% RSLogix 500 project AGEOVEN_NEW19.RSS, saved by version 12.00.00.00 %
PROJECT "UNTITLED"    % processor: type code 47 %

PROGRAM FILES
  LAD 2   3 rungs
  LAD 3   11 rungs
  LAD 4   8 rungs

DATA FILES
  O0 OUTPUT  9 elements
  I1 INPUT  9 elements
  S2 STATUS  83 elements
  B3 BINARY  1 elements
  T4 TIMER  1 elements
  C5 COUNTER  1 elements
  R6 CONTROL  1 elements
  N7 INTEGER  25 elements
  F8 FLOAT  2 elements

LADDER 2
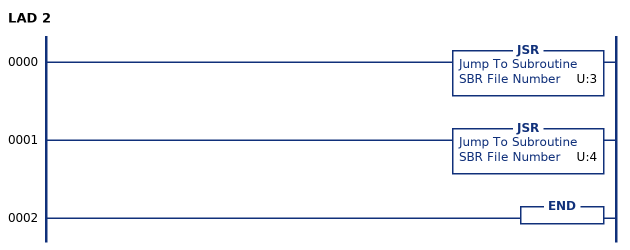
% Rung: 0 %
SOR JSR U:3 EOR
% Rung: 1 %
SOR JSR U:4 EOR
% Rung: 2 %
SOR END EOR

LADDER 3
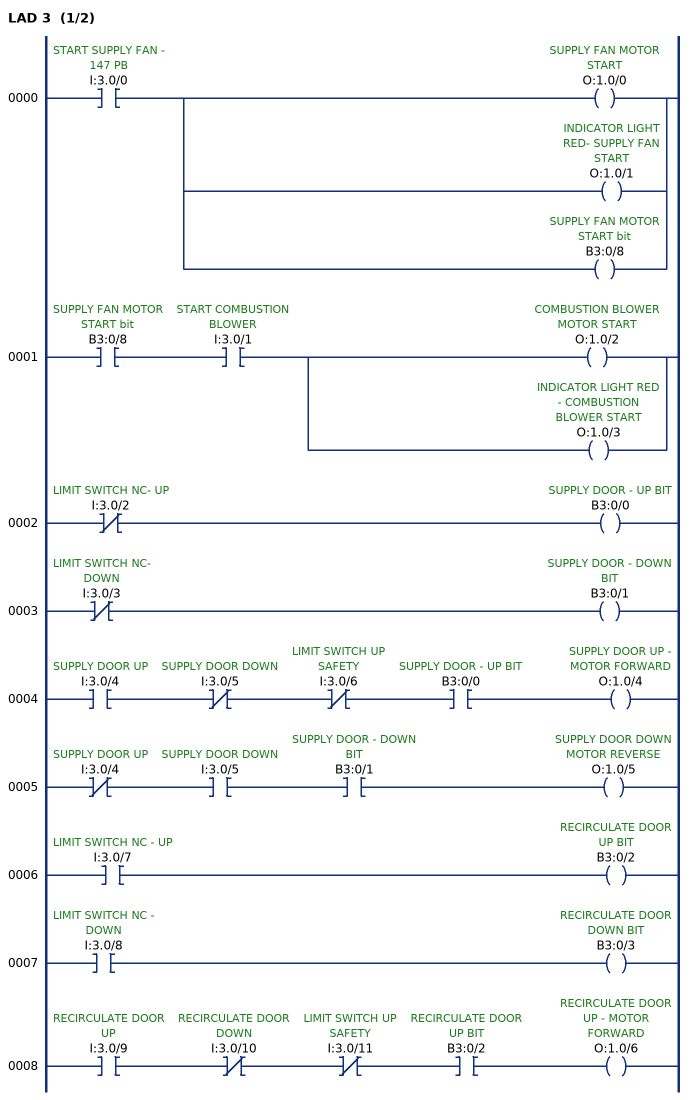
% Rung: 0 %
SOR XIC I:3.0/0 BST OTE O:1.0/0 NXB OTE O:1.0/1 NXB OTE B3:0/8 BND EOR
%   I:3.0/0  "START SUPPLY FAN - 147 PB" %
%   O:1.0/0  "SUPPLY FAN MOTOR START" %
%   O:1.0/1  "INDICATOR LIGHT RED- SUPPLY FAN START" %
%   B3:0/8  "SUPPLY FAN MOTOR START bit" %
% Rung: 1 %
SOR XIC B3:0/8 XIC I:3.0/1 BST OTE O:1.0/2 NXB OTE O:1.0/3 BND EOR
%   B3:0/8  "SUPPLY FAN MOTOR START bit" %
%   I:3.0/1  "START COMBUSTION BLOWER" %
%   O:1.0/2  "COMBUSTION BLOWER MOTOR START" %
%   O:1.0/3  "INDICATOR LIGHT RED - COMBUSTION BLOWER START" %
% Rung: 2 %  % edit flag set %
SOR XIO I:3.0/2 OTE B3:0/0 EOR
%   I:3.0/2  "LIMIT SWITCH NC- UP" %
%   B3:0/0  "SUPPLY DOOR - UP BIT" %
% Rung: 3 %  % edit flag set %
SOR XIO I:3.0/3 OTE B3:0/1 EOR
%   I:3.0/3  "LIMIT SWITCH NC- DOWN" %
%   B3:0/1  "SUPPLY DOOR - DOWN BIT" %
% Rung: 4 %
SOR XIC I:3.0/4 XIO I:3.0/5 XIO I:3.0/6 XIC B3:0/0 OTE O:1.0/4 EOR
%   I:3.0/4  "SUPPLY DOOR UP" %
%   I:3.0/5  "SUPPLY DOOR DOWN" %
%   I:3.0/6  "LIMIT SWITCH UP SAFETY" %
%   B3:0/0  "SUPPLY DOOR - UP BIT" %
%   O:1.0/4  "SUPPLY DOOR UP - MOTOR FORWARD" %
% Rung: 5 %
SOR XIO I:3.0/4 XIC I:3.0/5 XIC B3:0/1 OTE O:1.0/5 EOR
%   I:3.0/4  "SUPPLY DOOR UP" %
%   I:3.0/5  "SUPPLY DOOR DOWN" %
%   B3:0/1  "SUPPLY DOOR - DOWN BIT" %
%   O:1.0/5  "SUPPLY DOOR DOWN MOTOR REVERSE" %
% Rung: 6 %
SOR XIC I:3.0/7 OTE B3:0/2 EOR
%   I:3.0/7  "LIMIT SWITCH NC - UP" %
%   B3:0/2  "RECIRCULATE DOOR UP BIT" %
% Rung: 7 %
SOR XIC I:3.0/8 OTE B3:0/3 EOR
%   I:3.0/8  "LIMIT SWITCH NC - DOWN" %
%   B3:0/3  "RECIRCULATE DOOR DOWN BIT" %
% Rung: 8 %
SOR XIC I:3.0/9 XIO I:3.0/10 XIO I:3.0/11 XIC B3:0/2 OTE O:1.0/6 EOR
%   I:3.0/9  "RECIRCULATE DOOR UP" %
%   I:3.0/10  "RECIRCULATE DOOR DOWN" %
%   I:3.0/11  "LIMIT SWITCH UP SAFETY" %
%   B3:0/2  "RECIRCULATE DOOR UP BIT" %
%   O:1.0/6  "RECIRCULATE DOOR UP - MOTOR FORWARD" %

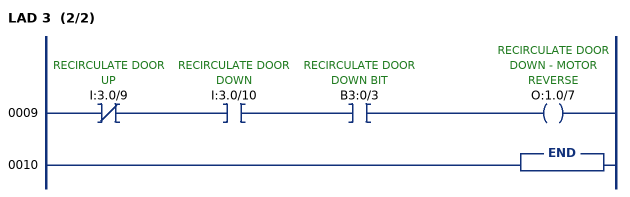
% Rung: 9 %
SOR XIO I:3.0/9 XIC I:3.0/10 XIC B3:0/3 OTE O:1.0/7 EOR
%   I:3.0/9  "RECIRCULATE DOOR UP" %
%   I:3.0/10  "RECIRCULATE DOOR DOWN" %
%   B3:0/3  "RECIRCULATE DOOR DOWN BIT" %
%   O:1.0/7  "RECIRCULATE DOOR DOWN - MOTOR REVERSE" %
% Rung: 10 %
SOR END EOR

LADDER 4
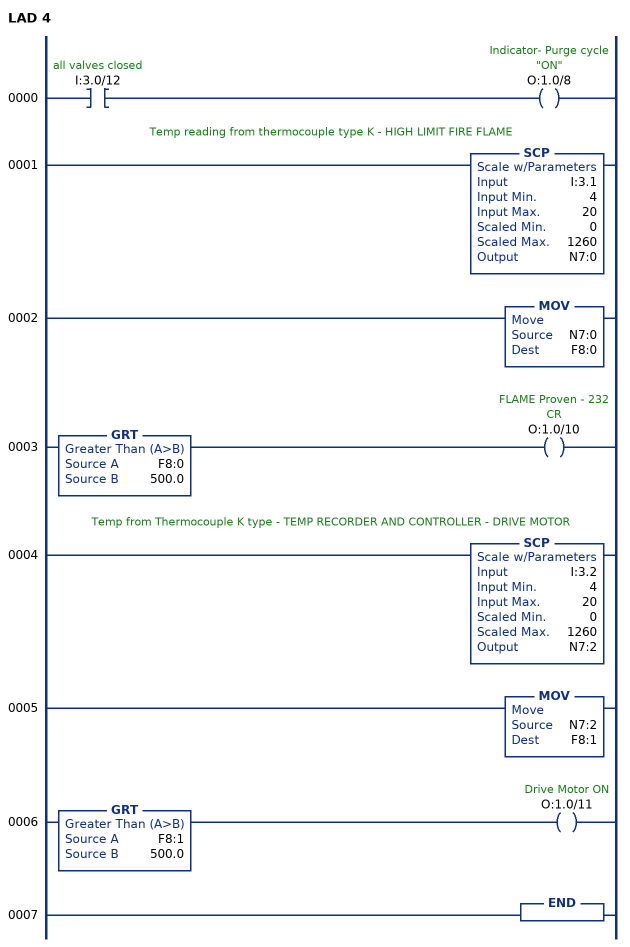
% Rung: 0 %
SOR XIC I:3.0/12 OTE O:1.0/8 EOR
%   I:3.0/12  "all valves closed" %
%   O:1.0/8  "Indicator- Purge cycle "ON"" %
% Rung: 1 %
% Temp reading from thermocouple type K - HIGH LIMIT FIRE FLAME %
SOR SCP I:3.1 4 20 0 1260 N7:0 EOR
%   I:3.1  "Thermocouple for tempretaure control" %
% Rung: 2 %
SOR MOV N7:0 F8:0 EOR
% Rung: 3 %
SOR GRT F8:0 500.0 OTE O:1.0/10 EOR
%   O:1.0/10  "FLAME Proven - 232 CR" %
% Rung: 4 %
% Temp from Thermocouple K type - TEMP RECORDER AND CONTROLLER - DRIVE MOTOR %
SOR SCP I:3.2 4 20 0 1260 N7:2 EOR
% Rung: 5 %
SOR MOV N7:2 F8:1 EOR
% Rung: 6 %
SOR GRT F8:1 500.0 OTE O:1.0/11 EOR
%   O:1.0/11  "Drive Motor ON" %
% Rung: 7 %
SOR END EOR

OTHER DOCUMENTED ADDRESSES
  I:3.3  "tHERMOCOUPLE INPUT"
  N7:1  "temp control"
  O:3.0/0  "SUPPLY FAN MOTOR"
  O:3.0/1  "SUPPLY FAN INDICATOR - RED"
  O:3.0/2  "COMBUSTION BLOWER MOTOR"
  O:3.0/3  "COMBUSTION BLOWER INDICATOR - RED"
  O:3.0/4  "SUPPLY DOOR UP- MOTOR FORWARD"
  O:3.0/5  "SUPPLY DOOR DOWN - MOTOR REVERSE"
  O:3.0/6  "RECIRCULATE DOOR UP - MOTOR FORWARD"
  O:3.0/7  "RECIRCULATE DOOR DOWN - MOTOR REVERSE"

DATA TABLE (non-zero values as saved)
DATA N7
% N7:0 % 0 0 500 0 500 0 0 1260 0 1250
% N7:10 % -200 0 0 0 0 0 0 0 0 0
